(* IEC 61131-3 sources: traffic-lights/PLC_TrafficLights/Class/ENVBase, 1 file *)

(* ---- ENVBase.st ---- *)
(*!
<Class
	Name               = "ENVBase"
	Revision           = "1.0"
	RealtimeTask       = "false"
	CyclicTask         = "false"
	BackgroundTask     = "false"
	Sigmatek           = "true"
	OSInterface        = "false"
	HighPriority       = "false"
	Automatic          = "false"
	UpdateMode         = "Prescan"
	SharedCommandTable = "true"
	Objectsize         = "(574,120)"
	Comment            = "just to get access to a change in the &#13;&#10;derived class">
	<Channels>
		<Server Name="sChangedVarName" Visualized="false" Initialize="false" WriteProtected="false" Retentive="false" Comment="to react on a change of the&#13;&#10;variable name"/>
		<Server Name="sChangedVarValue" Visualized="false" Initialize="false" WriteProtected="false" Retentive="false" Comment="to react on a change of the value"/>
		<Server Name="sStatus" Visualized="false" Initialize="false" WriteProtected="true" Retentive="false" Comment="state of executed Commands"/>
		<Client Name="ASCII_BIN" Required="true" Internal="true"/>
		<Client Name="EnvironmentVariableLib" Required="true" Internal="true"/>
	</Channels>
	<RevDoku>
		<Owner Company="Sigmatek" Author="hötant"/>
		<Dokumentation Revision="1.0" Date="2011-09-21" Author="hötant" Company="Sigmatek" Description="creation of class"/>
	</RevDoku>
	<Network Name="ENVBase">
		<!-- List of Components in this network -->
		<Components>
			<Object
				Name       = "ASCII_BIN"
				Class      = "ASCII_BIN"
				Position   = "(90,390)"
				Visualized = "true">
				<Channels>
					<Server Name="Obj_channel"/>
				</Channels>
			</Object>
			<Object
				Name       = "EnvironmentVariableLib"
				Class      = "ENVLib"
				Position   = "(90,180)"
				Visualized = "false">
				<Channels>
					<Server Name="ClassSvr"/>
				</Channels>
			</Object>
		</Components>
		<Comments>
		</Comments>
		<!-- List of Connections in this network -->
		<Connections>
			<Connection Source="this.EnvironmentVariableLib" Destination="EnvironmentVariableLib.ClassSvr"/>
			<Connection Source="this.ASCII_BIN" Destination="ASCII_BIN.Obj_channel"/>
		</Connections>
		<!-- Headerfiles -->
		<Options>
		</Options>
	</Network>
</Class>
*)
ENVBase : CLASS
  //Servers:
	sStatus 	: SvrChCmd_ENV_Status;
	sChangedVarName 	: SvrCh_DINT;
	sChangedVarValue 	: SvrCh_DINT;
  //Clients:
	EnvironmentVariableLib 	: CltChCmd_ENVLib;
	ASCII_BIN 	: CltChCmd_ASCII_BIN;
  //Variables:
  //Functions:
				//! <Function Comment="react on a user action.&#13;&#10;(e.g.: change of variable name ,..)&#13;&#10;" Name="SomethingChanged"/>
	FUNCTION VIRTUAL GLOBAL SomethingChanged
		VAR_INPUT
			Reaseon 	: DINT;			//! <Variable Comment="0.. Varialbe name changed&#13;&#10;1.. Sting Value Variable Changed&#13;&#10;2.. Numeric Value Changed" Name="SomethingChanged.Reaseon"/>
		END_VAR;

	FUNCTION VIRTUAL GLOBAL sChangedVarName::Write
		VAR_INPUT
			input (EAX) 	: DINT;
		END_VAR
		VAR_OUTPUT
			result (EAX) 	: DINT;
		END_VAR;

	FUNCTION VIRTUAL GLOBAL sChangedVarValue::Write
		VAR_INPUT
			input (EAX) 	: DINT;
		END_VAR
		VAR_OUTPUT
			result (EAX) 	: DINT;
		END_VAR;
  //Tables:
	FUNCTION @STD
		VAR_OUTPUT
			ret_code	: CONFSTATES;
		END_VAR;
	FUNCTION GLOBAL TAB @CT_;
END_CLASS;

#pragma using ASCII_BIN
#pragma using ENVLib

FUNCTION VIRTUAL GLOBAL ENVBase::sChangedVarName::Write
	VAR_INPUT
		input (EAX) 	: DINT;
	END_VAR
	VAR_OUTPUT
		result (EAX) 	: DINT;
	END_VAR

	SomethingChanged(Reaseon:=0);
 	result := input;

END_FUNCTION

FUNCTION VIRTUAL GLOBAL ENVBase::sChangedVarValue::Write
	VAR_INPUT
		input (EAX) 	: DINT;
	END_VAR
	VAR_OUTPUT
		result (EAX) 	: DINT;
	END_VAR

	SomethingChanged(Reaseon:=1);
 	result := input;

END_FUNCTION

#pragma warning(disable:73 )

FUNCTION VIRTUAL GLOBAL ENVBase::SomethingChanged
	VAR_INPUT
		Reaseon 	: DINT;
	END_VAR

END_FUNCTION

#pragma warning(default:73 )
